// TIA Portal V18 export
DATA_BLOCK "MES_CHeck_DB"   // DB111
// stored: AutoNumber false, InstanceOfName MES_CHeck, InstanceOfType FB
"MES_CHeck"
   // VAR
   //    Station_1 : "MES Check_fb";
   //    Station_2 : "MES Check_fb";
   //    Station_3 : "MES Check_fb";
   //    Station_4 : "MES Check_fb";
   //    Station_5 : "MES Check_fb";
   //    Station_6 : "MES Check_fb";
   //    Station_7 : "MES Check_fb";
   //    Station_8 : "MES Check_fb";
   // END_VAR
BEGIN
END_DATA_BLOCK
